{attribute 'qualified_only'}
{attribute 'strict'}
TYPE E_Popup :
(
	ePopupNone := 0,
	ePopupSafetyEs,
	ePopupStempelkissenWechseln,
	ePopup02,
	ePopup03,
	ePopup04,
	ePopupMax
);
END_TYPE

(* stored: Version 1.1.0.1
   DUT E_Popup: Id {138627db-24fc-4b7b-bda3-efe1e9c78bb1} *)
